// TIA Portal V20 export
DATA_BLOCK "IDB_LineA1"   // DB8
// stored: InstanceOfName LineA1.FB_LineA1, InstanceOfType FB, Namespace LineA1
"LineA1.FB_LineA1"
   // VAR
   //    "Conveyor_A1.1.1" : "Global.FB_Conveyor";
   //    "MABS_A1.1.1" : "Global.FB_MABS";
   //    "Transfer_A1.1.1" : "Global.FB_S300_tTransMode";
   // END_VAR
BEGIN
END_DATA_BLOCK
